{attribute 'Tc2GvlVarNames'}
{attribute 'strict'}
(* Pareggiatura Lastra da eseguire Prima del deposito *)
TYPE e_Stato_Pareggiatura_Lastra :
(
	PAREGGIATURA_DISABILITATA	:= 0, 
	PAREGGIATURA_DA_ESEGUIRE	:= 1, 
	PAREGGIATURA_ESEGUITA 		:= 2
);
END_TYPE

(* stored: Version 1.1.0.1, ProductVersion 3.1.4024.11
   EnumerationTextList e_Stato_Pareggiatura_Lastra: Id {ad1f6b98-fb70-47b0-a17e-260f46343f95} *)
